FUNCTION F_TestFunction : REAL
VAR_INPUT
END_VAR
VAR
END_VAR

F_TestFunction := 1337;

END_FUNCTION

(* stored: Version 1.1.0.1, ProductVersion 3.1.4024.12
   POU F_TestFunction: Id {158a3031-a16d-498d-b826-60c88cea8b08}, SpecialFunc None *)
